//SimpleObserver:
//Implements a simple observer which assumes the camera position is the true position of the robot whenever camera data arrives. Between new cam data
//odometry is used to correct the robots position. The cameras latency is also considered by correcting the arrived camera data with odometry based correction
//within the time interval of the latency. The observer is implemented in Simulink and is linked within this FB to abstract the implementation of the observer from the
//main control algorithm. Inside the Simulink model all coordinates are considered as world coordinates, following that the transformation of between robot and world coordinates 
//is implemented in ST.
FUNCTION_BLOCK SimpleObserverST
VAR_INPUT
	xCameraPose:	RobotPoseSimple;
	xVxRobot: 		LREAL;
	xVyRobot: 		LREAL;
	xOmegaRobot: 	LREAL;
	theta:			LREAL; //theta for I/O Lineraztion only explicitly Input for FF-Linearization
END_VAR

VAR_OUTPUT
	yObserverdPose: 	RobotPoseSimple;
END_VAR

VAR
	newCamDataArrived: BOOL;
	camDataOld, observerError, observedPosition, vWorld: RobotPoseSimple;
	pulseGenerator: TP;
	
	delayedCycles		AT%Q* 	: INT	:= 77;
	delayedPosition: ARRAY [0..140] OF RobotPoseSimple;
	
	
	K : ARRAY [0..2,0..2] OF LREAL 		:= [18, 0 ,0,
									  		0, 18, 0,
									  		0, 0, 18];
	
	// TEST
	//systime : NT_GetTime;
END_VAR

//transform roboter velocities into world velocities and pass them to Simulink
Robot2World( 
	vx_robot 	:= xVxRobot,
	vy_robot 	:= xVyRobot,
	omega_robot := xOmegaRobot,
	theta		:= yObserverdPose.theta,
	vx_world 	=> vWorld.x,
	vy_world  	=> vWorld.y,
	omega_world => vWorld.theta);
	
checkForNewCameraData();

//systime(START:=newCamDataArrived);	// TEST

delayPosition();
//if cam data arrived correct
IF newCamDataArrived THEN
	//calculate observer error
	observerError := SubtractRPS(xCameraPose,delayedPosition[delayedCycles]);
	//do the feedback correction
	observedPosition := AddRPS(observedPosition, ScaleRPS(c := Var_HAWIno.CONTROLLER_CYCLE_TIME, AddRPS(vWorld, MatrixTimesRPS(K, observerError))));
ELSE
	observedPosition := AddRPS(observedPosition, ScaleRPS(c := Var_HAWIno.CONTROLLER_CYCLE_TIME, vWorld));
END_IF


//set Outputs
yObserverdPose 	:= observedPosition;
camDataOld 		:= xCameraPose;

METHOD checkForNewCameraData : BOOL
VAR_INPUT
END_VAR
newCamDataArrived := (camDataOld.x <> xCameraPose.x OR camDataOld.y <> xCameraPose.y OR camDataOld.theta <> xCameraPose.theta) //cahnge in one of the positions
					 AND xCameraPose.x <> 0 AND xCameraPose.y <> 0;		//valid data
END_METHOD

METHOD PRIVATE delayPosition : BOOL
VAR_INPUT
END_VAR
VAR
	i: INT := 0;
END_VAR
FOR i := 0 TO delayedCycles-1 DO
	delayedPosition[i+1] := delayedPosition[i];
END_FOR
delayedPosition[0] := observedPosition;
END_METHOD

METHOD reset : BOOL
VAR_INPUT
END_VAR
VAR
	
END_VAR
observedPosition := xCameraPose;
END_METHOD

END_FUNCTION_BLOCK

(* stored: Version 1.1.0.1, ProductVersion 3.1.4024.11
   POU SimpleObserverST: Id {9bfb0c63-c7fa-4cc8-ba80-418e5355c9f5}, SpecialFunc None
   Method checkForNewCameraData: Id {f1cf2097-a90f-4703-bbdf-a246f17538d7}
   Method delayPosition: Id {1134d261-4292-4598-b780-bc2622c2593f}
   Method reset: Id {a72036aa-6b35-4ea4-8248-f4df1f99d19e} *)
